// TIA Portal project "level control" (V17)
// Vorlageprojekt für das Buch mit Zielsystem S7-1200

(* hardware
DEVICE "S7-1200-Station_1"  S7-1200 Station
   slot 0: "Baugruppenträger_0"  Rack  V1.0
   slot 1: "PLC_1"  CPU 1211C DC/DC/DC  6ES7 211-1AE40-0XB0  V4.1
*)

// ===== PLC "PLC_1"  CPU 1211C DC/DC/DC =====

VAR_GLOBAL   // PLC tag table "Standard-Variablentabelle"
   "start" AT %I0.0 : Bool;
   "reset" AT %I0.1 : Bool;
   "stop" AT %I0.2 : Bool;
   "FACTORY IO run" AT %I0.3 : Bool;
   "level meter" AT %ID30 : Real;
   "flow meter" AT %ID34 : Real;
   "setpoint" AT %ID38 : Real;
   "start light" AT %Q0.0 : Bool;
   "reset light" AT %Q0.1 : Bool;
   "stop light" AT %Q0.2 : Bool;
   "fill valve" AT %QD30 : Real;
   "discharge valve" AT %QD34 : Real;
   "sp" AT %QD38 : DInt;
   "pv" AT %QD42 : DInt;
   "Tag_3" AT %MD38 : Real;
   "Tag_1" AT %MD30 : Real;
   "Tag_2" AT %MD34 : DInt;
   "Tag_4" AT %MD42 : Real;
   "Tag_5" AT %MD40 : Real;
END_VAR

DATA_BLOCK "modes"   // DB2
{ S7_Optimized_Access := 'TRUE' }
VERSION : 0.1
   VAR
      "stop mode" : Bool;
      "start mode" : Bool;
      "reset mode" : Bool;
   END_VAR
BEGIN
END_DATA_BLOCK

FUNCTION "1 operation modes" : Void   // FC1, LAD
{ S7_Optimized_Access := 'TRUE' }
VERSION : 0.1
BEGIN

REGION Network 1: start mode
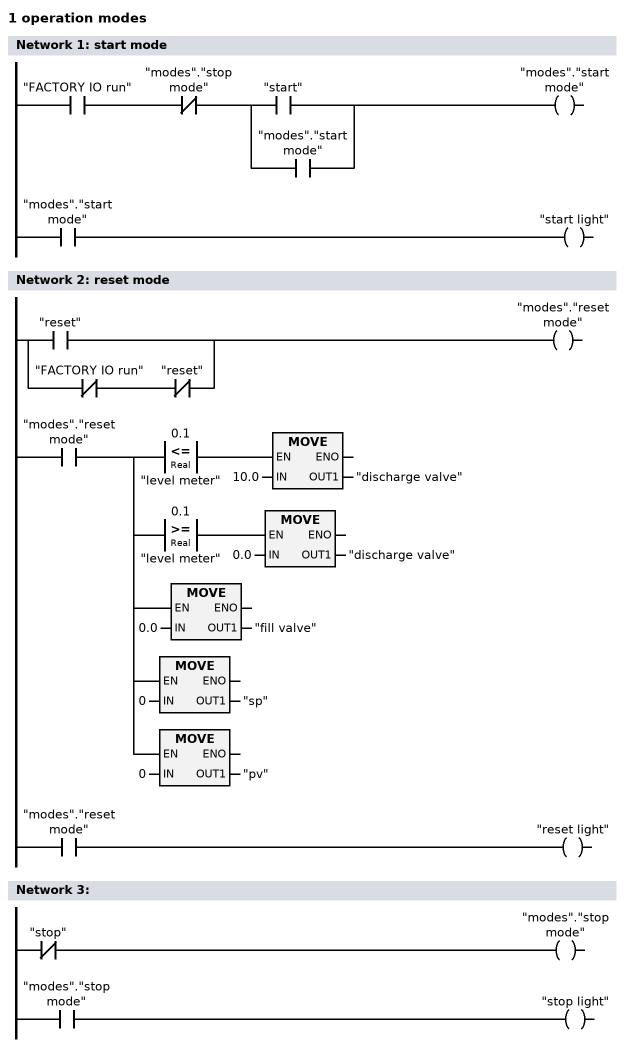
   RUNG wire#powerrail
      Contact( "FACTORY IO run" )
      I_Contact( "modes"."stop mode" )
      wire#w1
      Contact( "start" )
      wire#w2
      Coil( "modes"."start mode" )
   END_RUNG
   RUNG wire#w1
      Contact( "modes"."start mode" )
   END_RUNG wire#w2
   RUNG wire#powerrail
      Contact( "modes"."start mode" )
      Coil( "start light" )
   END_RUNG
   // the same network as SCL:
   "modes"."start mode" := "FACTORY IO run" AND NOT "modes"."stop mode" AND ("start" OR "modes"."start mode");
   "start light" := "modes"."start mode";
END_REGION

REGION Network 2: reset mode
   RUNG wire#powerrail
      Contact( "reset" )
      wire#w1
      Coil( "modes"."reset mode" )
   END_RUNG
   RUNG wire#powerrail
      I_Contact( "FACTORY IO run" )
      I_Contact( "reset" )
   END_RUNG wire#w1
   RUNG wire#powerrail
      Contact( "modes"."reset mode" )
      wire#w2
      { S7_Templates := "SrcType := Real" } LE_Contact(in1 := 0.1, in2 := "level meter")
      Move(in := 10.0, out1 => "discharge valve")
   END_RUNG
   RUNG wire#w2
      { S7_Templates := "SrcType := Real" } GE_Contact(in1 := 0.1, in2 := "level meter")
      Move(in := 0.0, out1 => "discharge valve")
   END_RUNG
   RUNG wire#w2
      Move(in := 0.0, out1 => "fill valve")
   END_RUNG
   RUNG wire#w2
      Move(in := 0, out1 => "sp")
   END_RUNG
   RUNG wire#w2
      Move(in := 0, out1 => "pv")
   END_RUNG
   RUNG wire#powerrail
      Contact( "modes"."reset mode" )
      Coil( "reset light" )
   END_RUNG
   // the same network as SCL:
   "modes"."reset mode" := "reset" OR (NOT "FACTORY IO run" AND NOT "reset");
   IF "modes"."reset mode" AND (0.1 <= "level meter") THEN "discharge valve" := 10.0; END_IF;
   IF "modes"."reset mode" AND (0.1 >= "level meter") THEN "discharge valve" := 0.0; END_IF;
   IF "modes"."reset mode" THEN
       "fill valve" := 0.0;
       "sp" := 0;
       "pv" := 0;
   END_IF;
   "reset light" := "modes"."reset mode";
END_REGION

REGION Network 3
   RUNG wire#powerrail
      I_Contact( "stop" )
      Coil( "modes"."stop mode" )
   END_RUNG
   RUNG wire#powerrail
      Contact( "modes"."stop mode" )
      Coil( "stop light" )
   END_RUNG
   // the same network as SCL:
   "modes"."stop mode" := NOT "stop";
   "stop light" := "modes"."stop mode";
END_REGION
END_FUNCTION

FUNCTION "2 step definition" : Void   // FC2, LAD
{ S7_Optimized_Access := 'TRUE' }
VERSION : 0.1
   VAR_TEMP   // added for the SCL form of the ladder/FBD networks
      _w1 : Bool;
   END_VAR
BEGIN

REGION Network 1: setare nivel dorit
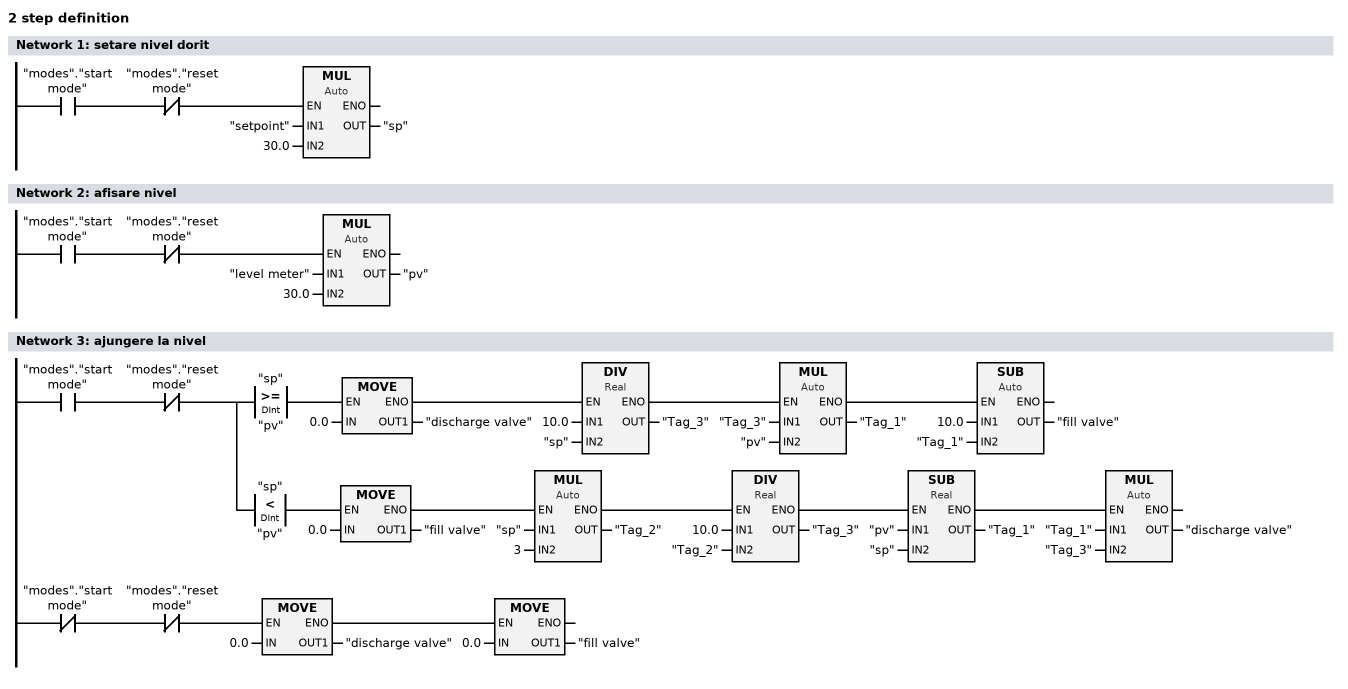
   RUNG wire#powerrail
      Contact( "modes"."start mode" )
      I_Contact( "modes"."reset mode" )
      Mul(in1 := "setpoint", in2 := 30.0, out => "sp")
   END_RUNG
   // the same network as SCL:
   IF "modes"."start mode" AND NOT "modes"."reset mode" THEN "sp" := "setpoint" * 30.0; END_IF;
END_REGION

REGION Network 2: afisare nivel
   RUNG wire#powerrail
      Contact( "modes"."start mode" )
      I_Contact( "modes"."reset mode" )
      Mul(in1 := "level meter", in2 := 30.0, out => "pv")
   END_RUNG
   // the same network as SCL:
   IF "modes"."start mode" AND NOT "modes"."reset mode" THEN "pv" := "level meter" * 30.0; END_IF;
END_REGION

REGION Network 3: ajungere la nivel
   RUNG wire#powerrail
      Contact( "modes"."start mode" )
      I_Contact( "modes"."reset mode" )
      wire#w1
      { S7_Templates := "SrcType := DInt" } GE_Contact(in1 := "sp", in2 := "pv")
      Move(in := 0.0, out1 => "discharge valve")
      { S7_Templates := "SrcType := Real" } Div(in1 := 10.0, in2 := "sp", out => "Tag_3")
      Mul(in1 := "Tag_3", in2 := "pv", out => "Tag_1")
      Sub(in1 := 10.0, in2 := "Tag_1", out => "fill valve")
   END_RUNG
   RUNG wire#w1
      { S7_Templates := "SrcType := DInt" } LT_Contact(in1 := "sp", in2 := "pv")
      Move(in := 0.0, out1 => "fill valve")
      Mul(in1 := "sp", in2 := 3, out => "Tag_2")
      { S7_Templates := "SrcType := Real" } Div(in1 := 10.0, in2 := "Tag_2", out => "Tag_3")
      { S7_Templates := "SrcType := Real" } Sub(in1 := "pv", in2 := "sp", out => "Tag_1")
      Mul(in1 := "Tag_1", in2 := "Tag_3", out => "discharge valve")
   END_RUNG
   RUNG wire#powerrail
      I_Contact( "modes"."start mode" )
      I_Contact( "modes"."reset mode" )
      Move(in := 0.0, out1 => "discharge valve")
      Move(in := 0.0, out1 => "fill valve")
   END_RUNG
   // the same network as SCL:
   #_w1 := "modes"."start mode" AND NOT "modes"."reset mode";
   IF #_w1 AND ("sp" >= "pv") THEN
       "discharge valve" := 0.0;
       "Tag_3" := 10.0 / "sp";
       "Tag_1" := "Tag_3" * "pv";
       "fill valve" := 10.0 - "Tag_1";
   END_IF;
   IF #_w1 AND ("sp" < "pv") THEN
       "fill valve" := 0.0;
       "Tag_2" := "sp" * 3;
       "Tag_3" := 10.0 / "Tag_2";
       "Tag_1" := "pv" - "sp";
       "discharge valve" := "Tag_1" * "Tag_3";
   END_IF;
   IF NOT "modes"."start mode" AND NOT "modes"."reset mode" THEN
       "discharge valve" := 0.0;
       "fill valve" := 0.0;
   END_IF;
END_REGION
END_FUNCTION

FUNCTION "MHJ-PLC-Lab-Function-S71200" : Void   // FC9000, SCL
{ S7_Optimized_Access := 'TRUE' }
VERSION : 0.1
   VAR_TEMP
      rdTimeReturn : Int;
      outputTime : DTL;
      SyncVal : Byte;
      forVal : Int;
      forVal_2 : Int;
      Value : Byte;
   END_VAR
   VAR CONSTANT
      CompVal : Byte := 16#34;
      Value_01 : Byte := 16#11;
      Value_01_DW : DWord := 16#A165_D992;
      Value_02_DW : DWord := 16#58BE_4401;
   END_VAR
BEGIN

   #Value:=PEEK(area := 16#82,
        dbNumber := 0,
        byteOffset := 511);
   #Value := #Value + 1;

   POKE(area := 16#82,
        dbNumber := 0,
        byteOffset := 511,
        value := #Value);

   POKE(area:=16#81,
        dbNumber:=0,
        byteOffset:=1016,
        value:=#Value_01_DW);
   POKE(area := 16#81,
        dbNumber := 0,
        byteOffset := 1020,
        value := #Value_02_DW);

   POKE(area := 16#81,
        dbNumber := 0,
        byteOffset := 511,
        value := B#16#00);

   FOR #forVal := 0 TO 120 DO
       FOR #forVal_2:=0 TO 10 DO
           #rdTimeReturn:=RD_SYS_T(#outputTime);
           #rdTimeReturn := WR_SYS_T(#outputTime);
           #rdTimeReturn := RD_SYS_T(#outputTime);
           #rdTimeReturn := WR_SYS_T(#outputTime);
       END_FOR;
       #SyncVal:= PEEK(area := 16#81,
                      dbNumber := 0,
                      byteOffset := 511);
       IF #SyncVal = #CompVal THEN
          GOTO M_1;
       END_IF;
   END_FOR;
   RETURN;

   M_1:
   POKE(area := 16#81,
        dbNumber := 0,
        byteOffset := 511,
        value := B#16#0);
END_FUNCTION

ORGANIZATION_BLOCK "Main"   // OB1, FBD, ProgramCycle
TITLE = "Main Program Sweep (Cycle)"
{ S7_Optimized_Access := 'TRUE' }
VERSION : 0.1
   VAR_INPUT
      Initial_Call : Bool;   // Initial call of this OB
      Remanence : Bool;   // =True, if remanent data are available
   END_VAR
BEGIN

REGION Network 1: Konnektierungsbaustein für PLC-Lab
   // Im Netzwerk 1 wird der Konnektierungsbaustein für PLC-Lab aufgerufen.
   // Dieser Aufruf darf nicht entfernt werden!
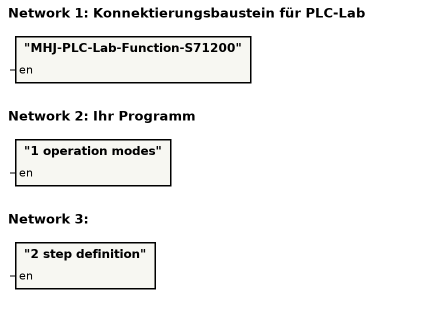
   "MHJ-PLC-Lab-Function-S71200"();
END_REGION

REGION Network 2: Ihr Programm
   // Schreiben Sie ab Netzwerk 2 Ihr Programm
   "1 operation modes"();
END_REGION

REGION Network 3
   "2 step definition"();
END_REGION
END_ORGANIZATION_BLOCK